(* CoDeSys 2.3 export: ATTR1_TU.EXP *)

(* Data type in Diag/Parameter *)
TYPE attr1_tu :
STRUCT
	MinValue_s16		: INT;
(*
	InputChannel_u16	: UINT;
	ListNumber_u16		: UINT;
	data_au8 			: ARRAY [1..2] OF USINT;
*)
END_STRUCT
END_TYPE
